(* PLC project Rasi_feeds_batching2.project, Automation Builder 2.7 - Basic Automation Builder 2.7 *)
(* stored: creationDateTime 2026-09-04T11:26:21.8292929, modificationDateTime 2026-09-04T10:44:56.4245457 *)

PROGRAM batching14
  VAR
    Auto_Ctrl : Auto_Batching_V14;
    Semi_Auto_Ctrl : Semi_Auto_Batching_V14;
    Auto_Complete : BOOL;
    Semi_Auto_Complete : BOOL;
    Auto_Err : INT;
    Auto_Msg : STRING;
    Semi_Auto_Err : INT;
    Semi_Auto_Msg : STRING;
    AutoBatchScale : MODRTUMAST;
    ModEnabler : BLINK;
    SamyakRaw : ARRAY[0..1] OF DINT;
    AutBatchRaw : ARRAY[0..1] OF DINT;
    SemAutoScale : MODRTUMAST;
    SemiAutoScaleRaw : ARRAY[0..1] OF DINT;
    AutoBatchSamyak : REAL;
    FB_Samyak_Multi_1 : FB_Samyak_Multi;
    FB_Samyak_Control_1 : FB_Samyak_Control;
    Run_PB_1 : BOOL;
    Next_Cycle_Start : BOOL;
    TP_1 : TP;
    TP_ON : BOOL;
    TP_Out : BOOL;
    TP_Et : TIME;
  END_VAR

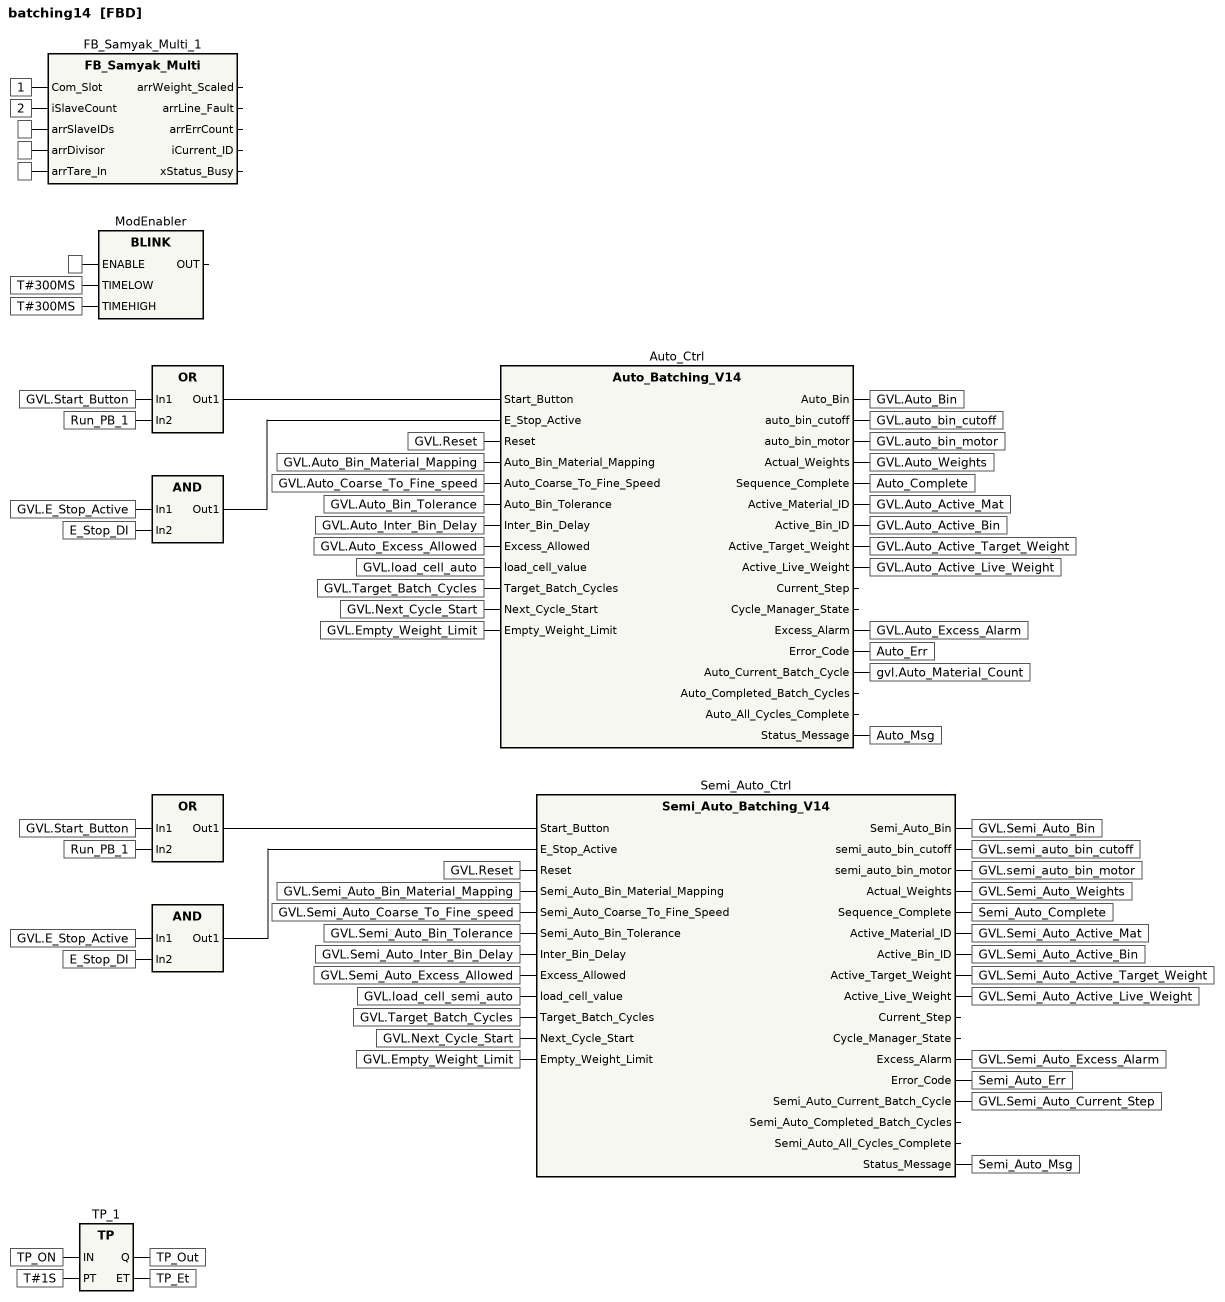
(* FBD diagram, written out as Structured Text *)
FB_Samyak_Multi_1(Com_Slot := 1, iSlaveCount := 2, arrSlaveIDs := , arrDivisor := , arrTare_In := );
ModEnabler(ENABLE := , TIMELOW := T#300MS, TIMEHIGH := T#300MS);
Auto_Ctrl(Start_Button := GVL.Start_Button OR Run_PB_1, E_Stop_Active := GVL.E_Stop_Active AND E_Stop_DI, Reset := GVL.Reset, Auto_Bin_Material_Mapping := GVL.Auto_Bin_Material_Mapping, Auto_Coarse_To_Fine_Speed := GVL.Auto_Coarse_To_Fine_speed, Auto_Bin_Tolerance := GVL.Auto_Bin_Tolerance, Inter_Bin_Delay := GVL.Auto_Inter_Bin_Delay, Excess_Allowed := GVL.Auto_Excess_Allowed, load_cell_value := GVL.load_cell_auto, Target_Batch_Cycles := GVL.Target_Batch_Cycles, Next_Cycle_Start := GVL.Next_Cycle_Start, Empty_Weight_Limit := GVL.Empty_Weight_Limit, auto_bin_cutoff => GVL.auto_bin_cutoff, auto_bin_motor => GVL.auto_bin_motor, Actual_Weights => GVL.Auto_Weights, Sequence_Complete => Auto_Complete, Active_Material_ID => GVL.Auto_Active_Mat, Active_Bin_ID => GVL.Auto_Active_Bin, Active_Target_Weight => GVL.Auto_Active_Target_Weight, Active_Live_Weight => GVL.Auto_Active_Live_Weight, Excess_Alarm => GVL.Auto_Excess_Alarm, Error_Code => Auto_Err, Auto_Current_Batch_Cycle => gvl.Auto_Material_Count, Status_Message => Auto_Msg);
GVL.Auto_Bin := Auto_Ctrl.Auto_Bin;
Semi_Auto_Ctrl(Start_Button := GVL.Start_Button OR Run_PB_1, E_Stop_Active := GVL.E_Stop_Active AND E_Stop_DI, Reset := GVL.Reset, Semi_Auto_Bin_Material_Mapping := GVL.Semi_Auto_Bin_Material_Mapping, Semi_Auto_Coarse_To_Fine_Speed := GVL.Semi_Auto_Coarse_To_Fine_speed, Semi_Auto_Bin_Tolerance := GVL.Semi_Auto_Bin_Tolerance, Inter_Bin_Delay := GVL.Semi_Auto_Inter_Bin_Delay, Excess_Allowed := GVL.Semi_Auto_Excess_Allowed, load_cell_value := GVL.load_cell_semi_auto, Target_Batch_Cycles := GVL.Target_Batch_Cycles, Next_Cycle_Start := GVL.Next_Cycle_Start, Empty_Weight_Limit := GVL.Empty_Weight_Limit, semi_auto_bin_cutoff => GVL.semi_auto_bin_cutoff, semi_auto_bin_motor => GVL.semi_auto_bin_motor, Actual_Weights => GVL.Semi_Auto_Weights, Sequence_Complete => Semi_Auto_Complete, Active_Material_ID => GVL.Semi_Auto_Active_Mat, Active_Bin_ID => GVL.Semi_Auto_Active_Bin, Active_Target_Weight => GVL.Semi_Auto_Active_Target_Weight, Active_Live_Weight => GVL.Semi_Auto_Active_Live_Weight, Excess_Alarm => GVL.Semi_Auto_Excess_Alarm, Error_Code => Semi_Auto_Err, Semi_Auto_Current_Batch_Cycle => GVL.Semi_Auto_Current_Step, Status_Message => Semi_Auto_Msg);
GVL.Semi_Auto_Bin := Semi_Auto_Ctrl.Semi_Auto_Bin;
TP_1(IN := TP_ON, PT := T#1S);
TP_Out := TP_1.Q;
TP_Et := TP_1.ET;
END_PROGRAM
